Yaskawa INFORM job: ARGPASS.JBI

/JOB
//NAME ARGPASS
//POS
///NPOS 0,0,0,0,0,0
//INST
///DATE 2026/05/06 10:37
///ATTR SC,RW
///GROUP1 RB1
NOP
CALL JOB:TOOLCHANGE ARGF5
END
